Staubli VAL3: page.pgx

public program page(string& menuname[], num index)
// set all the page
begin
  //
  //  PAGE
  //
  //,,,,,,,,,,,,,,,,,,,,,,,
  //  go home setting
  //,,,,,,,,,,,,,,,,,,,,,,,
  //
  //  HOME PAGE
  //
  //
  if index>=300 and index<=301
    title("< GO Home Setting Page > "+menuname)
  endIf

  //,,,,,,,,,,,,,,,,,,,,
  //  CYCLE
  //,,,,,,,,,,,,,,,,,,,,
  //  if index>=20 and index<=29
  //    title("< Production Page >")
  //  endIf
  //  if index>=200 and index<=209
  //    title("< Simulation >")
  //  endIf
  //  if index>=210 and index<=219
  //    title ("< Stepping Simulation >")
  //  endIf
  //
  //  MENU
  //
  menuname=""
  //,,,,,,,,,,,,,,,,,,,,
  //  KERNEL
  //,,,,,,,,,,,,,,,,,,,,
  switch index

    case 300
      // Programmer
      menuname="Test,,,,,Type,Delete,New"
    break
    case 301
      // Programmer
      menuname=",,,,,Type,Delete,New"
    break
    case 302
      // Programmer
      menuname="Mark,All,None,,,,<<,>>"
    break
    case 303
      // Programmer
      menuname="Here,Insert,Delete,,,,<<,>>"
    break
    case 304
      // Programmer
      menuname="Here,Insert,Delete,Move type,,,<<,>>"
    break

  endSwitch
end
